INTERFACE I_ExtensionVisitor

METHOD VisitExtension
VAR_INPUT
	VisitingExtension : I_Extension;
END_VAR
END_METHOD

END_INTERFACE

(* stored: Version 1.1.0.1, ProductVersion 3.1.4024.12
   Itf I_ExtensionVisitor: Id {85999d6c-b06f-4160-b5a9-bea6a13981be}
   Method VisitExtension: Id {7f8d01fe-e623-4511-926a-d6391bdbba9b} *)
